FUNCTION_BLOCK FB_TestSystem EXTENDS FB_SystemContinous
VAR_INPUT
END_VAR
VAR_OUTPUT
END_VAR
VAR	
	//OPC UA structures
	{attribute 'OPC.UA.DA' := '1'}
	localSetParameters : ST_TestSystemSetParameters;
	{attribute 'OPC.UA.DA' := '1'}
	localState : ST_TestSystemState;	

	//digital input
	bOperational 				AT %I*: BOOL;
	
	//digital output
	bSystemOperationOn 			AT %Q*: BOOL := FALSE;
		
	//components
	pumpGrundfosMagna3 			: FB_PumpGrundfosMagna3 := (fLowerSetPointLimit := 30, fUpperSetPointLimit := 100); 
	bStartPump					: BOOL := FALSE;
	fSetPointPump 				: REAL := 0;
	bAlgorithmPermissionPump 	: BOOL := TRUE;
	
	discreteValve				: FB_DiscreteValve;
	bOpenValve					: BOOL := FALSE;
	
	nInit						: BOOL := FALSE;
	

END_VAR

//set init values
IF(NOT nInit) THEN
	fSetPointAutomatic := 20;
	algorithmPermission := TRUE;
	nInit := TRUE;
END_IF

//start system methods
MAIN();
SetState();//set state values
SetOutput();//set output values

//pump
pumpGrundfosMagna3(
	bSetStatusOnAutomatic := bStartPump,
	fSetPointAutomatic := fSetPointPump,
	algorithmPermission := bAlgorithmPermissionPump
);

//discrete valve
discreteValve(
	bSetStatusOnAutomatic := bOpenValve,
	algorithmPermission := bAlgorithmPermissionPump);

METHOD PROTECTED  Operational : BOOL
VAR_INPUT
END_VAR
VAR_OUTPUT
	bSwitchToWorking : BOOL := FALSE;
END_VAR
bSystemOperationOn := TRUE;
bSwitchToWorking := TRUE;
END_METHOD

METHOD PROTECTED  RampDown : BOOL
VAR_INPUT
END_VAR
VAR_OUTPUT
	bRampDownFinished : BOOL := FALSE;
END_VAR
//turn system off
bSystemOperationOn := FALSE;

//turn pump off
bStartPump := FALSE;
fSetPointPump := 0;

bRampDownFinished := TRUE;
END_METHOD

METHOD PROTECTED  RampUp : BOOL
VAR_INPUT
END_VAR
VAR_OUTPUT
	bRampUpFinished : BOOL := FALSE;
END_VAR
VAR
END_VAR
//open valve
bOpenValve := TRUE;

//turn pump on
bStartPump := TRUE;
fSetPointPump := 100;

bRampUpFinished := TRUE;
END_METHOD

METHOD PRIVATE SetOutput : BOOL
VAR_INPUT
END_VAR
//set outputs from OPC UA
bSystemOperationOn := localSetParameters.bSystemOperationOn;
END_METHOD

METHOD PRIVATE SetState : BOOL
VAR_INPUT
END_VAR
//copy sensor values to OPC UA data struct


//copy states to OPC UA
controlState.bStatusOn := bSystemOperationOn;
END_METHOD

METHOD PROTECTED  StateCheck : BOOL
(* In this method the folowing elements of the actorState structrure have to be set if they are not set yet:
	bStatusOn 		: BOOL; //status on / off
	bError			: BOOL; //true if in error
	sErrorMessage	: STRING; //returns error message
	bWarning		: BOOL; //true if in warning
	sWarningMessage	: STRING; //returns warning message
	fOperatingPoint	: REAL; //current operating point
*)
VAR_INPUT
END_VAR
VAR
END_VAR
END_METHOD

METHOD PROTECTED  Working : BOOL
VAR_INPUT
END_VAR
VAR_OUTPUT
	bSwitchToOperational : BOOL := FALSE;
END_VAR
END_METHOD

END_FUNCTION_BLOCK

(* stored: Version 1.1.0.1, ProductVersion 3.1.4024.9
   POU FB_TestSystem: Id {7003cb31-5239-49d6-8372-83a96f9671f9}, SpecialFunc None
   Method Operational: Id {f0511b9d-ec63-4439-bedf-00ea55360bc5}
   Method RampDown: Id {b7b74ab3-d092-435e-8cae-255bb8b32b0c}
   Method RampUp: Id {f3784821-29fa-4a43-84ee-d8fad2aad1d8}
   Method SetOutput: Id {ed7a131a-a3a6-4bfc-ad29-fbe80c311f75}
   Method SetState: Id {c90130e8-67d0-4cc3-be94-df5af45a3604}
   Method StateCheck: Id {d5772649-a060-4f63-863c-5518172c4e38}
   Method Working: Id {108f57c1-42ce-4e97-b194-08b3f4031db8} *)
